(* Logix 5000 project; controller Savage_Saw vendor 1 type 14 code 154 rev 37.11; software revision 37.01; part 3 of 3 *)
(* tags used below, declared in another part *)
   Auto : BOOL;
   Axis : AxisData[3];
   AxisX_Gauge : ALIAS FOR Axis[0];
   AxisY_Traverse : ALIAS FOR Axis[1];
   AxisZ_RaiseLower : ALIAS FOR Axis[2];
   BladeChangeDone : BOOL;
   BumpDistanceDry : REAL;
   BumpDistanceWet : REAL;
   Fault : BOOL;
   GaugePotScale : REAL;
   GaugeVelocityHome : REAL;
   GaugeVelocityJogMax : REAL;
   HydReady : BOOL;
   HydRun : BOOL;
   HydRunning : BOOL;
   HydStart : BOOL;
   HydStop : BOOL;
   InAnPotGauge : ALIAS FOR Local:3:I.Ch1Data;
   inAnPotRaiseLower : ALIAS FOR Local:2:I.Ch1Data;
   inAnPotTraverse : ALIAS FOR Local:3:I.Ch0Data;
   inMS4CoolantPump : ALIAS FOR Local:1:I.Data.4;
   inSR1SafetyRelay : ALIAS FOR Local:1:I.Data.0;
   OilWarm : BOOL;
   outAnSpindleMotor : ALIAS FOR Local:5:O.Ch1Data;
   outAnSpindlePump : ALIAS FOR Local:5:O.Ch0Data;
   outCr01BrakeTraverse : ALIAS FOR RemoteHPU:4:O.0;
   outCr02BrakeGauge : ALIAS FOR RemoteHPU:4:O.1;
   outCr03BrakeRaiseLower : ALIAS FOR RemoteHPU:4:O.2;
   outCr04ClampAdvance : ALIAS FOR RemoteHPU:5:O.0;
   outCr05GageGripperAdvance : ALIAS FOR RemoteHPU:5:O.1;
   outCrlLaserLight : ALIAS FOR Local:8:O.Data.0;
   outLtaStackLtAmber : ALIAS FOR Local:8:O.Data.2;
   outLtgStackLtGreen : ALIAS FOR Local:8:O.Data.1;
   outLtrStackLtRed : ALIAS FOR Local:8:O.Data.3;
   outMs1HydrulicPump : ALIAS FOR Local:6:O.Data.0;
   outMs2LoopPump : ALIAS FOR Local:6:O.Data.1;
   outMs3HydraulicCoolFan : ALIAS FOR Local:6:O.Data.2;
   outMs4Coolant : ALIAS FOR Local:6:O.Data.3;
   outMs5SwarfPump : ALIAS FOR Local:7:O.Data.0;
   outMs6SwarfConveyor : ALIAS FOR Local:7:O.Data.1;
   RaiseLowerPotScale : REAL;
   RaiseLowerVelocityHome : REAL;
   RaiseLowerVelocityJogMax : REAL;
   RpmTarget : REAL;
   SpinCCWDemand : BOOL;
   SpinCWDemand : BOOL;
   SpinDemandFall : BOOL;
   SpindleMotorOutputScale : REAL;
   tbA1JogIn : BOOL;
   tbA1JogOut : BOOL;
   tbA2JogMinus : BOOL;
   tbA2JogPlus : BOOL;
   tbA3JogMinus : BOOL;
   tbA3JogPlus : BOOL;
   tbDryBump : BOOL;
   tbGaugeClamp : BOOL;
   tbGaugeUnclamp : BOOL;
   tbLaser : BOOL;
   tbMS2LoopPump : BOOL;
   tbMS3HydCoolingFan : BOOL;
   tbMS4CoolantPump : BOOL;
   tbMS5SwarfPump : BOOL;
   tbWetBump : BOOL;
   tbWorkClamp : BOOL;
   tbWorkUnclamp : BOOL;
   tbZeroGauge : BOOL;
   timerGaugeBrakeDelay : TIMER;
   timerRaiseLowerBrakeDelay : TIMER;
   timerTraverseBrakeDelay : TIMER;
   TraversePotScale : REAL;
   TraverseVelocityHome : REAL;
   TraverseVelocityJogMax : REAL;
   X_AutoCut : BOOL;
   X_Homing : BOOL;
   X_Manual : BOOL;
(* MainProgram, continued *)

ROUTINE X_Homing   (* ladder *)
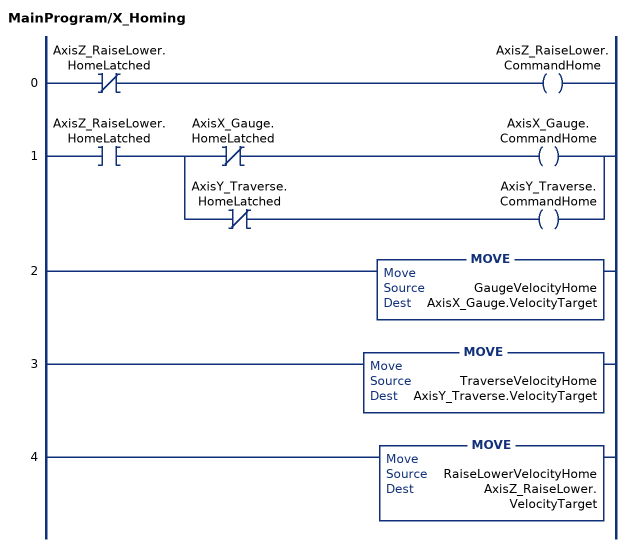
   0: XIO(AxisZ_RaiseLower.HomeLatched)OTE(AxisZ_RaiseLower.CommandHome);
   1: XIC(AxisZ_RaiseLower.HomeLatched)[XIO(AxisX_Gauge.HomeLatched) OTE(AxisX_Gauge.CommandHome) ,XIO(AxisY_Traverse.HomeLatched) OTE(AxisY_Traverse.CommandHome) ];
   2: MOVE(GaugeVelocityHome,AxisX_Gauge.VelocityTarget);
   3: MOVE(TraverseVelocityHome,AxisY_Traverse.VelocityTarget);
   4: MOVE(RaiseLowerVelocityHome,AxisZ_RaiseLower.VelocityTarget);
END_ROUTINE

ROUTINE X_Manual   (* ladder *)
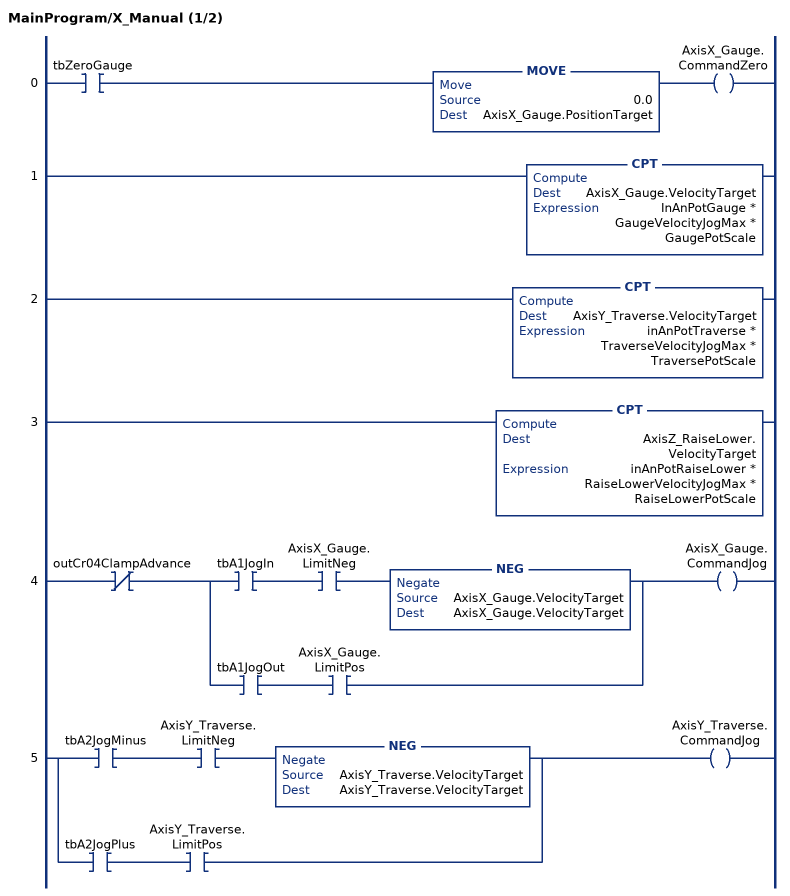
   0: XIC(tbZeroGauge)MOVE(0.0,AxisX_Gauge.PositionTarget)OTE(AxisX_Gauge.CommandZero);
   1: CPT(AxisX_Gauge.VelocityTarget,InAnPotGauge * GaugeVelocityJogMax * GaugePotScale);
   2: CPT(AxisY_Traverse.VelocityTarget,inAnPotTraverse * TraverseVelocityJogMax * TraversePotScale);
   3: CPT(AxisZ_RaiseLower.VelocityTarget,inAnPotRaiseLower * RaiseLowerVelocityJogMax * RaiseLowerPotScale);
   4: XIO(outCr04ClampAdvance)[XIC(tbA1JogIn) XIC(AxisX_Gauge.LimitNeg) NEG(AxisX_Gauge.VelocityTarget,AxisX_Gauge.VelocityTarget) ,XIC(tbA1JogOut) XIC(AxisX_Gauge.LimitPos) ]OTE(AxisX_Gauge.CommandJog);
   5: [XIC(tbA2JogMinus) XIC(AxisY_Traverse.LimitNeg) NEG(AxisY_Traverse.VelocityTarget,AxisY_Traverse.VelocityTarget) ,XIC(tbA2JogPlus) XIC(AxisY_Traverse.LimitPos) ]OTE(AxisY_Traverse.CommandJog);
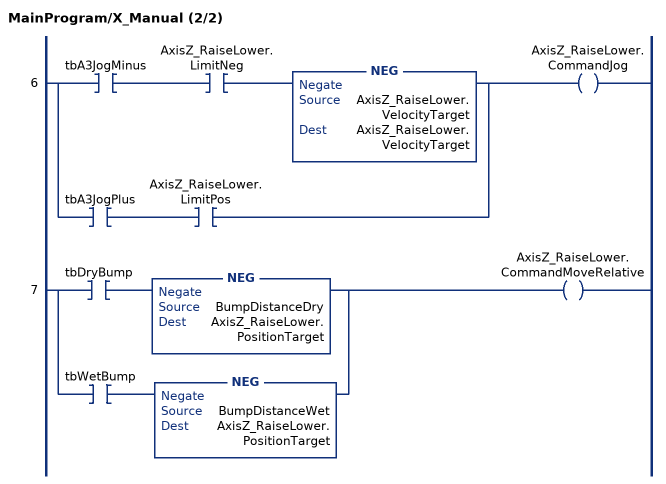
   6: [XIC(tbA3JogMinus) XIC(AxisZ_RaiseLower.LimitNeg) NEG(AxisZ_RaiseLower.VelocityTarget,AxisZ_RaiseLower.VelocityTarget) ,XIC(tbA3JogPlus) XIC(AxisZ_RaiseLower.LimitPos) ]OTE(AxisZ_RaiseLower.CommandJog);
   7: [XIC(tbDryBump) NEG(BumpDistanceDry,AxisZ_RaiseLower.PositionTarget) ,XIC(tbWetBump) NEG(BumpDistanceWet,AxisZ_RaiseLower.PositionTarget) ]OTE(AxisZ_RaiseLower.CommandMoveRelative);
END_ROUTINE
END_PROGRAM

PROGRAM Outputs   (* main routine Outputs *)
VAR
   iAxis : DINT;
   timerSwarfDelay : TIMER := (PRE := 1000);
END_VAR

ROUTINE Brakes   (* ladder *)
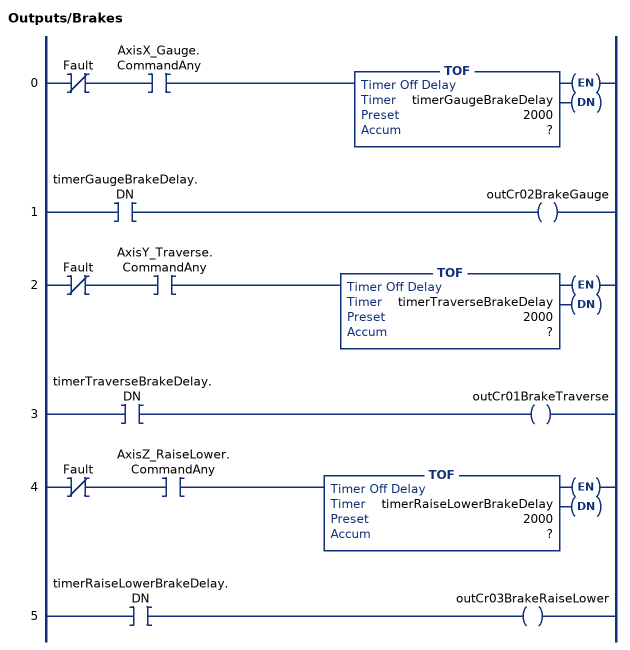
   0: XIO(Fault)XIC(AxisX_Gauge.CommandAny)TOF(timerGaugeBrakeDelay,?,?);
   1: XIC(timerGaugeBrakeDelay.DN)OTE(outCr02BrakeGauge);
   2: XIO(Fault)XIC(AxisY_Traverse.CommandAny)TOF(timerTraverseBrakeDelay,?,?);
   3: XIC(timerTraverseBrakeDelay.DN)OTE(outCr01BrakeTraverse);
   4: XIO(Fault)XIC(AxisZ_RaiseLower.CommandAny)TOF(timerRaiseLowerBrakeDelay,?,?);
   5: XIC(timerRaiseLowerBrakeDelay.DN)OTE(outCr03BrakeRaiseLower);
END_ROUTINE

ROUTINE Clamps   (* ladder *)
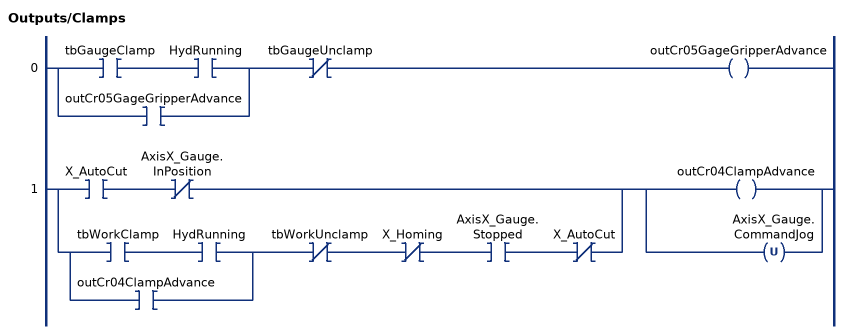
   0: [XIC(tbGaugeClamp) XIC(HydRunning) ,XIC(outCr05GageGripperAdvance) ]XIO(tbGaugeUnclamp)OTE(outCr05GageGripperAdvance);
   1: [XIC(X_AutoCut) XIO(AxisX_Gauge.InPosition) ,[XIC(tbWorkClamp) XIC(HydRunning) ,XIC(outCr04ClampAdvance) ] XIO(tbWorkUnclamp) XIO(X_Homing) XIC(AxisX_Gauge.Stopped) XIO(X_AutoCut) ][OTE(outCr04ClampAdvance) ,OTU(AxisX_Gauge.CommandJog) ];
END_ROUTINE

ROUTINE Coolant   (* ladder *)
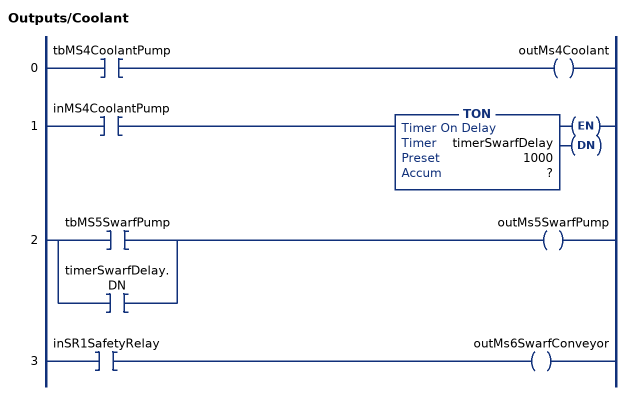
   0: XIC(tbMS4CoolantPump)OTE(outMs4Coolant);
   1: XIC(inMS4CoolantPump)TON(timerSwarfDelay,?,?);
   2: [XIC(tbMS5SwarfPump) ,XIC(timerSwarfDelay.DN) ]OTE(outMs5SwarfPump);
   3: XIC(inSR1SafetyRelay)OTE(outMs6SwarfConveyor);
END_ROUTINE

ROUTINE Hydraulics   (* ladder *)
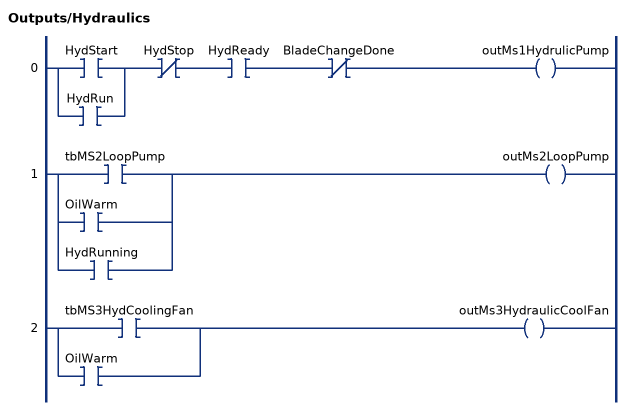
   0: [XIC(HydStart) ,XIC(HydRun) ]XIO(HydStop)XIC(HydReady)XIO(BladeChangeDone)OTE(outMs1HydrulicPump);
   1: [XIC(tbMS2LoopPump) ,XIC(OilWarm) ,XIC(HydRunning) ]OTE(outMs2LoopPump);
   2: [XIC(tbMS3HydCoolingFan) ,XIC(OilWarm) ]OTE(outMs3HydraulicCoolFan);
END_ROUTINE

ROUTINE Outputs   (* ladder *)
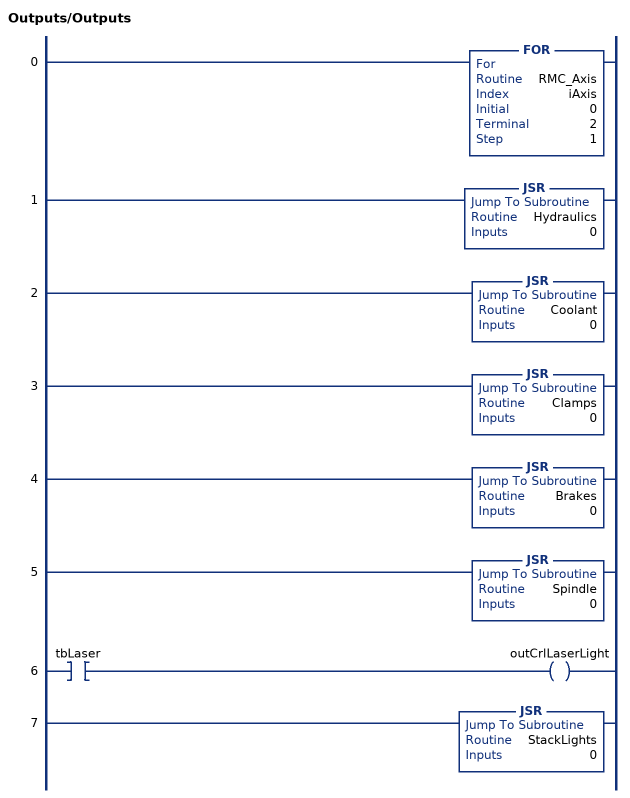
   0: FOR(RMC_Axis,iAxis,0,2,1);
   1: JSR(Hydraulics,0);
   2: JSR(Coolant,0);
   3: JSR(Clamps,0);
   4: JSR(Brakes,0);
   5: JSR(Spindle,0);
   6: XIC(tbLaser)OTE(outCrlLaserLight);
   7: JSR(StackLights,0);
END_ROUTINE

ROUTINE RMC_Axis   (* ladder *)
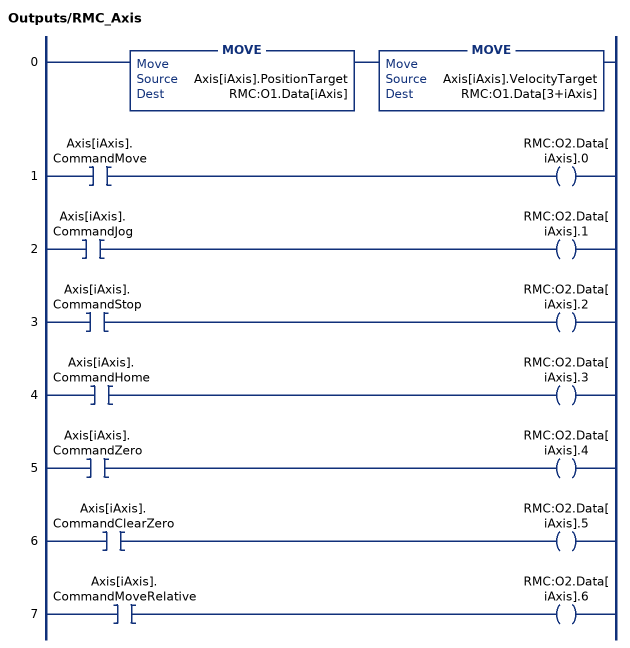
   0: MOVE(Axis[iAxis].PositionTarget,RMC:O1.Data[iAxis])MOVE(Axis[iAxis].VelocityTarget,RMC:O1.Data[3+iAxis]);
   1: XIC(Axis[iAxis].CommandMove)OTE(RMC:O2.Data[iAxis].0);
   2: XIC(Axis[iAxis].CommandJog)OTE(RMC:O2.Data[iAxis].1);
   3: XIC(Axis[iAxis].CommandStop)OTE(RMC:O2.Data[iAxis].2);
   4: XIC(Axis[iAxis].CommandHome)OTE(RMC:O2.Data[iAxis].3);
   5: XIC(Axis[iAxis].CommandZero)OTE(RMC:O2.Data[iAxis].4);
   6: XIC(Axis[iAxis].CommandClearZero)OTE(RMC:O2.Data[iAxis].5);
   7: XIC(Axis[iAxis].CommandMoveRelative)OTE(RMC:O2.Data[iAxis].6);
END_ROUTINE

ROUTINE Spindle   (* ladder *)
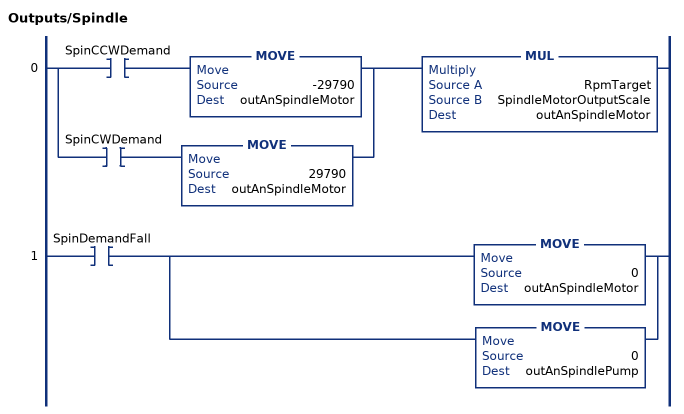
   0: [XIC(SpinCCWDemand) MOVE(-29790,outAnSpindleMotor) ,XIC(SpinCWDemand) MOVE(29790,outAnSpindleMotor) ]MUL(RpmTarget,SpindleMotorOutputScale,outAnSpindleMotor);
   1: XIC(SpinDemandFall)[MOVE(0,outAnSpindleMotor) ,MOVE(0,outAnSpindlePump) ];
END_ROUTINE

ROUTINE StackLights   (* ladder *)
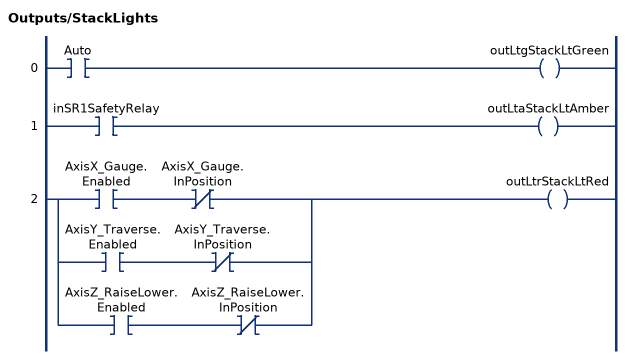
   0: XIC(Auto)OTE(outLtgStackLtGreen);
   1: XIC(inSR1SafetyRelay)OTE(outLtaStackLtAmber);
   2: [XIC(AxisX_Gauge.Enabled) XIO(AxisX_Gauge.InPosition) ,XIC(AxisY_Traverse.Enabled) XIO(AxisY_Traverse.InPosition) ,XIC(AxisZ_RaiseLower.Enabled) XIO(AxisZ_RaiseLower.InPosition) ]OTE(outLtrStackLtRed);
END_ROUTINE
END_PROGRAM
